INTERFACE IMachine EXTENDS ZApplication.IUnit

END_INTERFACE

(* stored: Version 1.1.0.1
   Itf IMachine: Id {b0710145-60c9-4dd6-8f74-4b8f09ab1990} *)
